TYPE DUT_SENSOR_DATAS_5 :
UNION
	data_lreal:REAL;
	data_byte:ARRAY[0..3] OF BYTE;
END_UNION
END_TYPE

(* stored: Version 1.1.0.1, ProductVersion 3.1.4024.6
   DUT DUT_SENSOR_DATAS_5: Id {dd0f1298-2008-4170-a0c8-16af0dd98140} *)
